FUNCTION_BLOCK SeqTransfer (* Basic Function Block Type *)
  (* Standard: 61499-2 *)
  (* Version 0.0, 2/16/2024, midxav, Template *)
  PACKAGE Main;
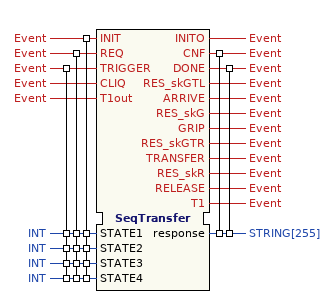
  EVENT_INPUT
    INIT WITH STATE1, STATE2, STATE3, STATE4; (* Initialization Request *)
    REQ WITH STATE1, STATE2, STATE3, STATE4; (* Normal Execution Request *)
    TRIGGER WITH STATE1, STATE2, STATE3, STATE4;
    CLIQ;
    T1out;
  END_EVENT
  EVENT_OUTPUT
    INITO; (* Initialization Confirm *)
    CNF WITH response; (* Execution Confirmation *)
    DONE WITH response;
    RES_skGTL;
    ARRIVE;
    RES_skG;
    GRIP;
    RES_skGTR;
    TRANSFER;
    RES_skR;
    RELEASE;
    T1;
  END_EVENT
  VAR_INPUT
    STATE1 : INT;
    STATE2 : INT;
    STATE3 : INT;
    STATE4 : INT;
  END_VAR
  VAR_OUTPUT
    response : STRING[255];
  END_VAR
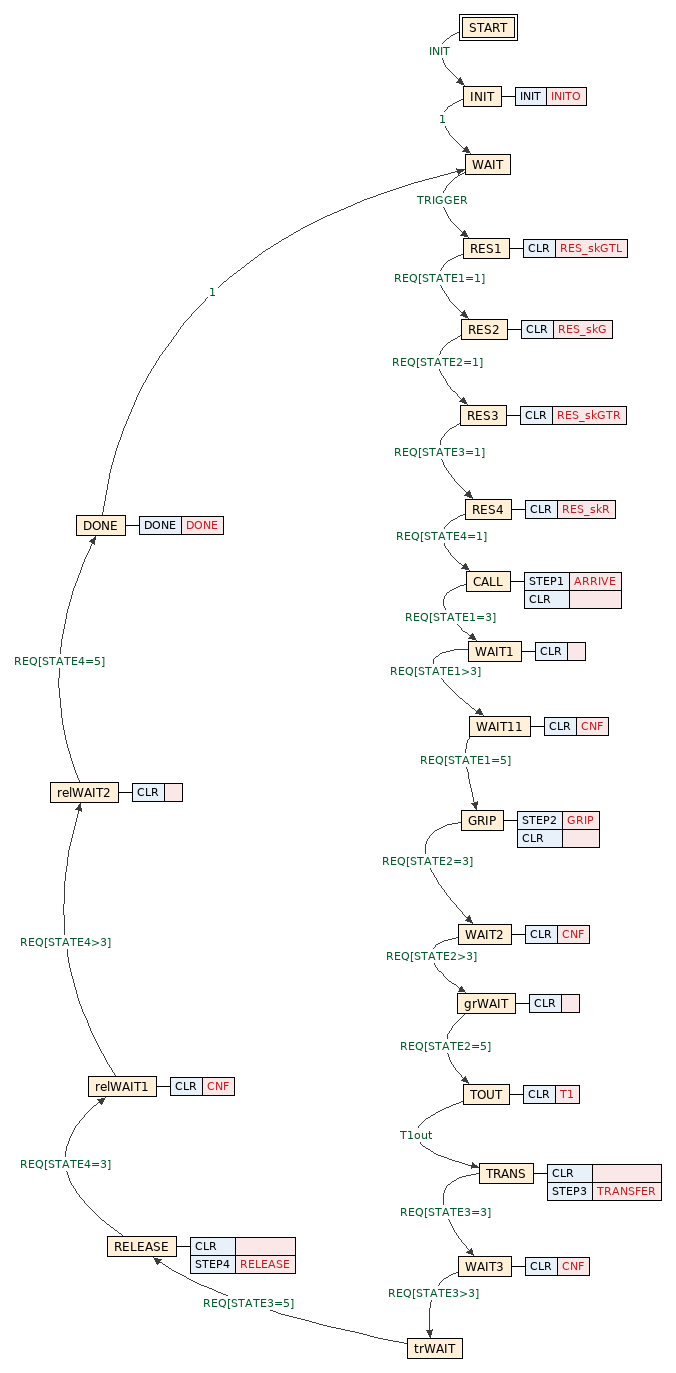
  EC_STATES
    START; (* Initial State *)
    INIT : INIT -> INITO; (* Initialization *)
    DONE : DONE -> DONE;
    WAIT;
    CALL : STEP1 -> ARRIVE, CLR;
    GRIP : STEP2 -> GRIP, CLR;
    WAIT1 : CLR;
    TRANS : CLR, STEP3 -> TRANSFER;
    WAIT2 : CLR -> CNF;
    RELEASE : CLR, STEP4 -> RELEASE;
    WAIT3 : CLR -> CNF;
    relWAIT1 : CLR -> CNF;
    WAIT11 : CLR -> CNF;
    RES1 : CLR -> RES_skGTL;
    RES2 : CLR -> RES_skG;
    RES3 : CLR -> RES_skGTR;
    RES4 : CLR -> RES_skR;
    TOUT : CLR -> T1;
    grWAIT : CLR;
    trWAIT;
    relWAIT2 : CLR;
  END_STATES
  EC_TRANSITIONS
    START TO INIT := INIT;
    DONE TO WAIT := 1;
    INIT TO WAIT := 1;
    WAIT1 TO WAIT11 := REQ[STATE1>3];
    CALL TO WAIT1 := REQ[STATE1=3];
    WAIT2 TO grWAIT := REQ[STATE2>3];
    GRIP TO WAIT2 := REQ[STATE2=3];
    WAIT3 TO trWAIT := REQ[STATE3>3];
    TRANS TO WAIT3 := REQ[STATE3=3];
    WAIT TO RES1 := TRIGGER;
    relWAIT1 TO relWAIT2 := REQ[STATE4>3];
    RELEASE TO relWAIT1 := REQ[STATE4=3];
    WAIT11 TO GRIP := REQ[STATE1=5];
    RES4 TO CALL := REQ[STATE4=1];
    RES1 TO RES2 := REQ[STATE1=1];
    RES2 TO RES3 := REQ[STATE2=1];
    RES3 TO RES4 := REQ[STATE3=1];
    TOUT TO TRANS := T1out;
    grWAIT TO TOUT := REQ[STATE2=5];
    trWAIT TO RELEASE := REQ[STATE3=5];
    relWAIT2 TO DONE := REQ[STATE4=5];
  END_TRANSITIONS
  ALGORITHM INIT IN ST: (* Initialization algorithm *)
;
  END_ALGORITHM
  ALGORITHM GoToMag IN ST:
;
  END_ALGORITHM
  ALGORITHM DONE IN ST:
response:='WP TRANSFERRED';
  END_ALGORITHM
  ALGORITHM ERROR IN ST:
response:='ALREADY AT LEFT SIDE';
TRIGGER:=FALSE;
  END_ALGORITHM
  ALGORITHM STEP1 IN ST:
response:='ARM MOVES LEFT';
TRIGGER:=FALSE;
  END_ALGORITHM
  ALGORITHM STEP2 IN ST:
response:='GRIPPING WP';
TRIGGER:=FALSE;
  END_ALGORITHM
  ALGORITHM STEP3 IN ST:
response:='ARM MOVES RIGHT';
TRIGGER:=FALSE;
  END_ALGORITHM
  ALGORITHM STEP4 IN ST:
response:='RELEASING WP';
TRIGGER:=FALSE;
  END_ALGORITHM
  ALGORITHM CLR IN ST:
REQ:=FALSE;
  END_ALGORITHM
END_FUNCTION_BLOCK
